FUNCTION_BLOCK CM_Servo EXTENDS CM_Base //IMPLEMENTS I_Servo
VAR_INPUT
	i_refAxis : REFERENCE TO Tc2_MC2.AXIS_REF;
	i_mcHomingMode : Tc2_MC2.MC_HomingMode := Tc2_MC2.MC_HomingMode.MC_Direct;
	i_mcBufferMode : Tc2_MC2.MC_BufferMode := Tc2_MC2.MC_BufferMode.MC_Aborting;
	i_bIclkForward : BOOL := TRUE; //TRUE = interlocked
	i_bIclkBackward : BOOL := TRUE; //TRUE = interlocked
	
	//--i_ref_setting : REFERENCE TO ST_PositioningProfile;
	i_ref_setting : REFERENCE TO ST_SettingsServo;
	
	
	i_ref_eCtrlState : REFERENCE TO E_CtrlState;
END_VAR

VAR
	fbPower : Tc2_MC2.MC_Power;
	fbReset : Tc2_MC2.MC_Reset;
	fbHome : Tc2_MC2.MC_Home;
	fbJog : Tc2_MC2.MC_Jog;
	fbMoveAbsolute : Tc2_MC2.MC_MoveAbsolute;
	fbStop : Tc2_MC2.MC_Stop;

	s_bStaAbsPosBusy : BOOL;
	s_fSetTargetPosition : LREAL;
	
	// Inputs
	I_bEnable AT %I* : BOOL; //Enable from safety controller
	I_bDetReferenceSwitch AT %I* : BOOL; //Reference-/home switch
	I_bDetLimitSwitchPositive AT %I* : BOOL; //Limit switch positive-/CW- direction
	I_bDetLimitSwitchNegative AT %I* : BOOL; //Limit switch negative-/CCW- direction
	
	//Properties
	s_bStatus : BOOL;
	s_bDone : BOOL; 
	s_bBusy : BOOL; 
	s_bActive : BOOL; 
	s_bCommandAborted : BOOL;
	s_bError : BOOL; 
	s_nErrorID : UDINT;
	
	//Requests
	s_bReqNcStop : BOOL;
	s_bReqNcReset : BOOL;
	s_bReqNcHome : BOOL;
	s_bReqNcJog : BOOL;
	s_bReqNcMoveAbs : BOOL;	
	
	// States
	s_bStaEnabled : BOOL;
	s_bStaReferenceSwitch : BOOL;
	s_bStaLimitSwitchPositive : BOOL;
	s_bStaLimitSwitchNegative : BOOL;
	
	s_bStaEnabledControl : BOOL;
	s_bStaEnabledForward : BOOL;
	s_bStaEnabledBackward : BOOL;
	s_bStaReady : BOOL;
	s_bStaHomed : BOOL;
	s_bStaStandstill : BOOL;
	s_bStaMoving : BOOL;
	s_bStaAtPosition : BOOL;
	s_bStaDriveError : BOOL;
	s_bStaWarning : BOOL;
	
	s_bIclkForward : BOOL;
	s_bIclkBackward : BOOL;
	s_sInterlockedReasonForward : STRING; //External interlocked reason for clarifying reason
	s_sInterlockedReasonBackward : STRING; //External interlocked reason for clarifying reason
	
	// Setpoints
	s_fTargetSpeed : LREAL; // Target speed [mm/s]
	
	
	// Alarms
	s_fbAlarmHandlerDriveError : FB_AlarmHandler;
	s_fbAlarmHandlerStartMotorNotAllowed : FB_AlarmHandler;
	s_fbAlarmHandlerMotorForwardInterlocked : FB_AlarmHandler;
	s_fbAlarmHandlerMotorBackwardInterlocked : FB_AlarmHandler;
	
	s_fbAlarmHandlerNotEnabled : FB_AlarmHandler;
	s_fbAlarmHandlerLimitPositiveReached : FB_AlarmHandler;
	s_fbAlarmHandlerLimitNegativeReached : FB_AlarmHandler;
	
	s_errDriveError : BOOL;
	s_wrnMotorForwardInterlocked : BOOL;
	s_wrnMotorBackwardInterlocked : BOOL;
	
	//Hmi
	s_fbHmiBtnHome : FB_HmiBtn;
	s_fbHmiBtnJogPos : FB_HmiBtn;
	s_fbHmiBtnJogNeg : FB_HmiBtn;
	s_fbHmiBtnMoveAbs : FB_HmiBtn;
	//--s_fbHmiBtnPower	: FB_HmiBtn;
	s_fbHmiBtnReset	: FB_HmiBtn;
	s_fbHmiBtnStop: FB_HmiBtn;
	
	s_fbHmiLedEnabledControl : FB_HmiLed;
	s_fbHmiLedEnabledForward : FB_HmiLed;
	s_fbHmiLedEnabledBackward : FB_HmiLed;
	s_fbHmiLedReady : FB_HmiLed;
	s_fbHmiLedHomed : FB_HmiLed;
	s_fbHmiLedStandstill : FB_HmiLed;
	s_fbHmiLedMoving : FB_HmiLed;
	s_fbHmiLedAtPosition : FB_HmiLed;
	s_fbHmiLedDriveError : FB_HmiLed;
	
	//Sequence
	s_eSeqNcTask : E_SeqServo;
	s_fbSeqNcTaskControl : FB_SeqControl;
	s_mcDirection : Tc2_MC2.MC_Direction;
END_VAR


fbPower(
	Axis := i_refAxis,
	Enable := I_bEnable,
	Enable_Positive := I_bDetLimitSwitchPositive,
	Enable_Negative := I_bDetLimitSwitchNegative,
	Override := 100.0,
	BufferMode := TC2_MC2.MC_BufferMode.MC_Aborting,
	Options := ,
	Status => s_bStatus,
	Busy => s_bBusy,
	Active => s_bActive,
	Error => s_bError,
	ErrorID => s_nErrorID);

SUPER^();

METHOD PROTECTED _m_Alarms : BOOL
VAR
	s_bPositiveDirection : BOOL; 
END_VAR

IF NOT SUPER^._m_Alarms() THEN
	RETURN;
END_IF

// Set error bits
s_errDriveError := (i_bReqEnable AND s_bStaDriveError) AND NOT(i_bCmdReset);

// Interlock warnings
s_bPositiveDirection := (i_refAxis.NcToPlc.ActVelo > 0);

IF s_bIclkForward AND NOT(s_bStaStandstill) AND s_bPositiveDirection THEN	
	s_wrnMotorForwardInterlocked := TRUE;
	
	m_Stop(
		i_fDec := i_ref_setting.fStopDec,
		i_fJrk := i_ref_setting.fStopJrk);
	
ELSIF NOT(s_bIclkForward) OR i_bCmdReset THEN
	s_wrnMotorForwardInterlocked := FALSE;
END_IF

IF s_bIclkBackward AND NOT(s_bStaStandstill) AND NOT(s_bPositiveDirection) THEN
	s_wrnMotorBackwardInterlocked := TRUE;
	
	m_Stop(
		i_fDec := i_ref_setting.fStopDec,
		i_fJrk := i_ref_setting.fJogJrk);
		
ELSIF NOT(s_bIclkBackward) OR i_bCmdReset THEN
	s_wrnMotorBackwardInterlocked := FALSE;
END_IF

// Alarm Handlers
s_fbAlarmHandlerDriveError(
	i_bStaActive := s_errDriveError,
	i_sAlarmText := CONCAT(i_sCmName, CONCAT(': Drive - has error: ', UDINT_TO_STRING(i_refAxis.NcToPlc.ErrorCode))));
	
s_fbAlarmHandlerMotorForwardInterlocked(
	i_bStaActive := s_wrnMotorForwardInterlocked,
	i_sAlarmText := CONCAT(i_sCmName, CONCAT(': Motor - interlocked to move forward, Reason: ',CONCAT(s_sInterlockedReasonForward, '.'))));
	
s_fbAlarmHandlerMotorBackwardInterlocked(
	i_bStaActive := s_wrnMotorBackwardInterlocked,
	i_sAlarmText := CONCAT(i_sCmName, CONCAT(': Motor - interlocked to move backward, Reason: ',CONCAT(s_sInterlockedReasonBackward, '.'))));

s_fbAlarmHandlerNotEnabled(
	i_bStaActive := NOT(s_bStaEnabled));
	
s_fbAlarmHandlerLimitPositiveReached(
	i_bStaActive := NOT(s_bStaLimitSwitchPositive));
	
s_fbAlarmHandlerLimitNegativeReached(
	i_bStaActive := NOT(s_bStaLimitSwitchNegative));	
	
// Alarm collector	
s_bStaError := 
	s_fbAlarmHandlerDriveError.q_bStaActive;

// Warning collector
s_bStaWarning := 
	s_fbAlarmHandlerMotorForwardInterlocked.q_bStaActive
	OR s_fbAlarmHandlerMotorBackwardInterlocked.q_bStaActive
	OR s_fbAlarmHandlerNotEnabled.q_bStaActive
	OR s_fbAlarmHandlerLimitPositiveReached.q_bStaActive
	OR s_fbAlarmHandlerLimitNegativeReached.q_bStaActive;
	
_m_Alarms := TRUE;
END_METHOD

METHOD PROTECTED _m_Devices : BOOL
VAR
	sTcDirection : Tc2_MC2.MC_Direction;
END_VAR
IF NOT SUPER^._m_Devices() THEN
	RETURN;
END_IF

s_bStaEnabledControl := s_bStaEnabled AND fbPower.Status;
s_bStaEnabledForward := s_bStaLimitSwitchPositive;
s_bStaEnabledBackward := s_bStaLimitSwitchNegative;

s_bStaReady := i_refAxis.NcToPlc.StateDWord.0;
s_bStaHomed := i_refAxis.NcToPlc.StateDWord.1;
s_bStaStandstill := i_refAxis.NcToPlc.StateDWord.2;
s_bStaMoving := NOT(i_refAxis.NcToPlc.StateDWord.2);
s_bStaAtPosition := i_refAxis.NcToPlc.StateDWord.4;
s_bStaDriveError := i_refAxis.NcToPlc.StateDWord.31;

s_fbSeqNcTaskControl(
	i_nSeqStep := s_eSeqNcTask, 
	i_sStepName := TO_STRING(s_eSeqNcTask), 
	i_bCmdReset := FALSE, 
	i_bStaError := FALSE);

	IF s_bReqNcStop THEN 
		s_eSeqNcTask := E_SeqServo.STOP;
	END_IF		
	
CASE s_eSeqNcTask OF

	E_SeqServo.IDLE:
		
		IF s_bReqNcStop THEN 
			s_eSeqNcTask := E_SeqServo.STOP;
		ELSIF s_bReqNcReset THEN
			s_eSeqNcTask := E_SeqServo.RESET;
		ELSIF s_bReqNcHome THEN
			s_eSeqNcTask := E_SeqServo.HOME;
		ELSIF s_bReqNcJog THEN
			s_eSeqNcTask := E_SeqServo.JOG;
		ELSIF s_bReqNcMoveAbs THEN
			s_eSeqNcTask := E_SeqServo.MOVE_ABS;	
		END_IF
		
	E_SeqServo.STOP:
		IF fbStop.Done THEN
			s_bReqNcStop := FALSE;
			s_eSeqNcTask := E_SeqServo.IDLE;
		END_IF
			
	E_SeqServo.RESET:
		IF fbReset.Done THEN
			s_bReqNcReset := FALSE;
			s_eSeqNcTask := E_SeqServo.IDLE;
		END_IF
			
	E_SeqServo.HOME:
		IF fbHome.Done THEN
			s_bReqNcHome := FALSE;
			s_eSeqNcTask := E_SeqServo.IDLE;
		END_IF
	
	E_SeqServo.JOG:
			IF NOT(s_fbHmiBtnJogPos.p_bStaBtn AND s_fbHmiBtnJogNeg.p_bStaBtn) OR fbJog.Error OR fbJog.CommandAborted THEN
				s_bReqNcJog := FALSE;
				s_eSeqNcTask := E_SeqServo.IDLE;
			END_IF
			
	E_SeqServo.MOVE_ABS:
		IF fbMoveAbsolute.Done OR fbMoveAbsolute.Error OR fbMoveAbsolute.CommandAborted THEN
			s_bReqNcMoveAbs := FALSE;
			s_eSeqNcTask := E_SeqServo.IDLE;
		END_IF
		
END_CASE

fbStop(
	Axis := i_refAxis,
	Execute := s_bReqNcStop,
	Deceleration := i_ref_setting.fStopDec,
	Jerk := i_ref_setting.fStopJrk,
	Options := ,
	Done => s_bDone,
	Busy => s_bBusy,
	Active => s_bActive,
	CommandAborted => s_bCommandAborted,
	Error => s_bError,
	ErrorID => s_nErrorID);

fbReset(
	Axis := i_refAxis,
	Execute := s_bReqNcReset,
	Done => s_bDone,
	Busy => s_bBusy,
	Error => s_bError,
	ErrorID => s_nErrorID);

fbHome(
	Axis := i_refAxis,
	Execute := s_bReqNcHome,
	Position := i_ref_setting.fHomeOffset,
	HomingMode := i_mcHomingMode,
	BufferMode := i_mcBufferMode,
	Options := ,
	bCalibrationCam := I_bDetReferenceSwitch,
	Done => s_bDone,
	Busy => s_bBusy,
	Active => s_bActive,
	CommandAborted => s_bCommandAborted,
	Error => s_bError,
	ErrorID => s_nErrorID);	
	
fbJog(
	Axis := i_refAxis,
	JogForward := s_fbHmiBtnJogPos.p_bStaBtn,
	JogBackwards := s_fbHmiBtnJogNeg.p_bStaBtn,
	Mode := MC_JOGMODE_STANDARD_SLOW,
	Position := ,
	Velocity := i_ref_setting.fJogVel,
	Acceleration := i_ref_setting.fJogAcc,
	Deceleration := i_ref_setting.fJogDec,
	Jerk := i_ref_setting.fJogJrk,
	Done => s_bDone,
	Busy => s_bBusy,
	Active => s_bActive,
	CommandAborted => s_bCommandAborted,
	Error => s_bError,
	ErrorID => s_nErrorID);
	
IF (i_eCtrlMode <> E_CtrlMode.AUTOMATIC) AND (i_eCtrlMode <> E_CtrlMode.MANUAL) THEN
	//--fbMoveAbsolute.Position := i_ref_setting.fAbsPosPos;
	fbMoveAbsolute.Position := s_fSetTargetPosition;
	fbMoveAbsolute.Velocity := i_ref_setting.fAbsPosVel;
	fbMoveAbsolute.Acceleration := i_ref_setting.fAbsPosAcc;
	fbMoveAbsolute.Deceleration := i_ref_setting.fAbsPosDec;
	fbMoveAbsolute.Jerk := i_ref_setting.fAbsPosJrk;
ELSE
	; //positining settings are written from the sequence (this could be different in each case)
END_IF
	
fbMoveAbsolute(
	Axis := i_refAxis,
	Execute := s_bReqNcMoveAbs, 
	Position := ,
	Velocity := ,
	Acceleration := ,
	Deceleration := ,
	Jerk := ,
	BufferMode := i_mcBufferMode,
	Options := ,
	Done => s_bDone,
	Busy => s_bBusy,
	Active => s_bActive,
	CommandAborted => s_bCommandAborted,
	Error => s_bError,
	ErrorID => s_nErrorID);
	
_m_Devices := TRUE;
END_METHOD

METHOD PROTECTED _m_Hmi : BOOL

IF NOT SUPER^._m_Hmi() THEN
	RETURN;
END_IF

//Buttons
s_fbHmiBtnHome();
s_fbHmiBtnJogPos();
s_fbHmiBtnJogNeg();
s_fbHmiBtnMoveAbs();
//--s_fbHmiBtnPower();
s_fbHmiBtnReset();
s_fbHmiBtnStop();

//Leds
s_fbHmiLedEnabledControl(i_bStaLed := s_bStaEnabledControl);
s_fbHmiLedEnabledForward(i_bStaLed := s_bStaEnabledForward);
s_fbHmiLedEnabledBackward(i_bStaLed := s_bStaEnabledBackward);
s_fbHmiLedReady(i_bStaLed := s_bStaReady);
s_fbHmiLedHomed(i_bStaLed := s_bStaHomed);
s_fbHmiLedStandstill(i_bStaLed := s_bStaStandstill);
s_fbHmiLedMoving(i_bStaLed := s_bStaMoving);
s_fbHmiLedAtPosition(i_bStaLed := s_bStaAtPosition);
s_fbHmiLedDriveError(i_bStaLed := s_bStaDriveError);

IF __ISVALIDREF(i_ref_eCtrlState) THEN
	//MAINTENANCE-mode is running
	IF (i_eCtrlMode = E_CtrlMode.MAINTENANCE) AND (i_ref_eCtrlState = E_CtrlState.RUNNING) THEN
		s_fbHmiBtnHome.p_bStaVisible := TRUE;
		s_fbHmiBtnHome.p_bStaEnabled := i_bReqEnable AND s_bStaEnabledControl AND s_bStaStandstill;	

		s_fbHmiBtnJogPos.p_bStaVisible := TRUE;
		s_fbHmiBtnJogPos.p_bStaEnabled := i_bReqEnable AND s_bStaEnabledControl AND s_bStaEnabledForward AND NOT(i_bIclkForward) AND NOT(s_bStaAbsPosBusy);
		
		s_fbHmiBtnJogNeg.p_bStaVisible := TRUE;
		s_fbHmiBtnJogNeg.p_bStaEnabled := i_bReqEnable AND s_bStaEnabledControl AND s_bStaEnabledBackward AND NOT(i_bIclkBackward) AND NOT(s_bStaAbsPosBusy);
	
		s_fbHmiBtnMoveAbs.p_bStaVisible := TRUE;
		s_fbHmiBtnMoveAbs.p_bStaEnabled := i_bReqEnable AND s_bStaEnabledControl AND s_bStaEnabledForward AND s_bStaEnabledBackward AND s_bStaStandstill AND s_bStaHomed AND NOT(i_bIclkForward) AND NOT(i_bIclkBackward);
		
		//--s_fbHmiBtnPower.p_bStaVisible := TRUE;
		//--s_fbHmiBtnPower.p_bStaEnabled := TRUE;
		
		s_fbHmiBtnReset.p_bStaVisible := TRUE;
		s_fbHmiBtnReset.p_bStaEnabled := TRUE;
		
		s_fbHmiBtnStop.p_bStaVisible := TRUE;
		s_fbHmiBtnStop.p_bStaEnabled := TRUE;
		
		//Maintenance commands from buttons
		IF s_fbHmiBtnStop.p_osrBtnPress THEN
			s_bReqNcStop := TRUE;
		END_IF
		
		IF s_fbHmiBtnReset.p_osrBtnPress THEN
			s_bReqNcReset := TRUE;
		END_IF
		
		IF s_fbHmiBtnHome.p_osrBtnPress THEN
			s_bReqNcHome := TRUE;
		END_IF
		
		IF s_fbHmiBtnJogNeg.p_osrBtnPress THEN
			s_mcDirection := Tc2_MC2.MC_Direction.MC_Negative_Direction;
			s_bReqNcJog := TRUE;
		END_IF
		
		IF s_fbHmiBtnJogPos.p_osrBtnPress THEN
			s_mcDirection := Tc2_MC2.MC_Direction.MC_Positive_Direction;
			s_bReqNcJog := TRUE;
		END_IF
		
		IF s_fbHmiBtnMoveAbs.p_osrBtnPress THEN
			s_bReqNcMoveAbs := TRUE;
		END_IF
		
	//other-mode	
	ELSE
		s_fbHmiBtnHome.p_bStaVisible := FALSE;
		s_fbHmiBtnHome.p_bStaEnabled := FALSE;
		
		s_fbHmiBtnJogPos.p_bStaVisible := FALSE;
		s_fbHmiBtnJogPos.p_bStaEnabled := FALSE;
		
		s_fbHmiBtnJogNeg.p_bStaVisible := FALSE;
		s_fbHmiBtnJogNeg.p_bStaEnabled := FALSE;
		
		s_fbHmiBtnMoveAbs.p_bStaVisible := FALSE;
		s_fbHmiBtnMoveAbs.p_bStaEnabled := FALSE;
		
		//--s_fbHmiBtnPower.p_bStaVisible := FALSE;
		//--s_fbHmiBtnPower.p_bStaEnabled := FALSE;
		
		s_fbHmiBtnReset.p_bStaVisible := FALSE;
		s_fbHmiBtnReset.p_bStaEnabled := FALSE;
		
		s_fbHmiBtnStop.p_bStaVisible := FALSE;
		s_fbHmiBtnStop.p_bStaEnabled := FALSE;
	END_IF
END_IF
	
_m_Hmi := TRUE;
END_METHOD

METHOD PROTECTED _m_Init : BOOL

IF NOT SUPER^._m_Init() THEN
	RETURN;
END_IF

//Alarm Config
// Alarm Handlers
s_fbAlarmHandlerDriveError.i_eAlarmLevel := E_AlarmLevel.Alarm;
s_fbAlarmHandlerMotorForwardInterlocked.i_eAlarmLevel := E_AlarmLevel.Warning;
s_fbAlarmHandlerMotorBackwardInterlocked.i_eAlarmLevel := E_AlarmLevel.Warning;
s_fbAlarmHandlerNotEnabled.i_eAlarmLevel := E_AlarmLevel.Warning;
s_fbAlarmHandlerNotEnabled.i_sAlarmText := CONCAT(i_sCmName, ' - Not enabled');
s_fbAlarmHandlerLimitPositiveReached.i_eAlarmLevel := E_AlarmLevel.Warning;
s_fbAlarmHandlerLimitPositiveReached.i_sAlarmText := CONCAT(i_sCmName, ' - Limits witch positvie reached');
s_fbAlarmHandlerLimitNegativeReached.i_eAlarmLevel := E_AlarmLevel.Warning;
s_fbAlarmHandlerLimitNegativeReached.i_sAlarmText := CONCAT(i_sCmName, ' - Limits witch negative reached');

//Hmi 
	//Buttons
	s_fbHmiBtnHome.p_eButtontype := E_HmiButtonType.PUSHBUTTON;
	s_fbHmiBtnHome.p_bStaVisible := FALSE;
	s_fbHmiBtnHome.p_bStaEnabled := FALSE;		
	s_fbHmiBtnHome.p_sBtnText := 'Home';
	
	s_fbHmiBtnJogPos.p_eButtontype := E_HmiButtonType.PUSHBUTTON;
	s_fbHmiBtnJogPos.p_bStaVisible := FALSE;
	s_fbHmiBtnJogPos.p_bStaEnabled := FALSE;		
	s_fbHmiBtnJogPos.p_sBtnText := 'Jog Positive';
	
	s_fbHmiBtnJogNeg.p_eButtontype := E_HmiButtonType.PUSHBUTTON;
	s_fbHmiBtnJogNeg.p_bStaVisible := FALSE;
	s_fbHmiBtnJogNeg.p_bStaEnabled := FALSE;		
	s_fbHmiBtnJogNeg.p_sBtnText := 'Jog Negative';
	
	s_fbHmiBtnMoveAbs.p_eButtontype := E_HmiButtonType.PUSHBUTTON;
	s_fbHmiBtnMoveAbs.p_bStaVisible := FALSE;
	s_fbHmiBtnMoveAbs.p_bStaEnabled := FALSE;		
	s_fbHmiBtnMoveAbs.p_sBtnText := 'Move Absolute';
	
	//--s_fbHmiBtnPower.p_eButtontype := E_HmiButtonType.PUSHBUTTON;
	//--s_fbHmiBtnPower.p_bStaVisible := FALSE;
	//--s_fbHmiBtnPower.p_bStaEnabled := FALSE;		
	//--s_fbHmiBtnPower.p_sBtnText := 'Enable';

	s_fbHmiBtnReset.p_eButtontype := E_HmiButtonType.PUSHBUTTON;
	s_fbHmiBtnReset.p_bStaVisible := FALSE;
	s_fbHmiBtnReset.p_bStaEnabled := FALSE;		
	s_fbHmiBtnReset.p_sBtnText := 'Reset';
	
	s_fbHmiBtnReset.p_eButtontype := E_HmiButtonType.PUSHBUTTON;
	s_fbHmiBtnReset.p_bStaVisible := FALSE;
	s_fbHmiBtnReset.p_bStaEnabled := FALSE;		
	s_fbHmiBtnReset.p_sBtnText := 'Reset';
	
	s_fbHmiBtnStop.p_eButtontype := E_HmiButtonType.PUSHBUTTON;
	s_fbHmiBtnStop.p_bStaVisible := FALSE;
	s_fbHmiBtnStop.p_bStaEnabled := FALSE;		
	s_fbHmiBtnStop.p_sBtnText := 'Stop';
	
	//Leds
	s_fbHmiLedEnabledControl.p_bStaVisible := FALSE;
	s_fbHmiLedEnabledControl.p_sToHmiDescriptionLed := 'Enabled Control';
	
	s_fbHmiLedEnabledForward.p_bStaVisible := FALSE;
	s_fbHmiLedEnabledForward.p_sToHmiDescriptionLed := 'Enabled Forward';
	
	s_fbHmiLedEnabledBackward.p_bStaVisible := FALSE;
	s_fbHmiLedEnabledBackward.p_sToHmiDescriptionLed := 'Enabled Backward';
	
	s_fbHmiLedReady.p_bStaVisible := FALSE;
	s_fbHmiLedReady.p_sToHmiDescriptionLed := 'Ready';
	
	s_fbHmiLedHomed.p_bStaVisible := FALSE;
	s_fbHmiLedHomed.p_sToHmiDescriptionLed := 'Homed';
	
	s_fbHmiLedStandstill.p_bStaVisible := FALSE;
	s_fbHmiLedStandstill.p_sToHmiDescriptionLed := 'Standstill';
	
	s_fbHmiLedMoving.p_bStaVisible := FALSE;
	s_fbHmiLedMoving.p_sToHmiDescriptionLed := 'Moving';

	s_fbHmiLedAtPosition.p_bStaVisible := FALSE;
	s_fbHmiLedAtPosition.p_sToHmiDescriptionLed := 'At Position';
	
	s_fbHmiLedDriveError.p_bStaVisible := FALSE;
	s_fbHmiLedDriveError.p_sToHmiDescriptionLed := 'Drive Error';
	
_m_Init := TRUE;
END_METHOD

METHOD PROTECTED _m_Inputs : BOOL

IF NOT SUPER^._m_Inputs() THEN
	RETURN;
END_IF

s_bReqNcReset := i_bCmdReset; 

s_bStaEnabled := I_bEnable;
s_bStaReferenceSwitch := I_bDetReferenceSwitch;
s_bStaLimitSwitchPositive := I_bDetLimitSwitchPositive;
s_bStaLimitSwitchNegative := I_bDetLimitSwitchNegative;

s_bIclkForward := i_bIclkForward;
s_bIclkBackward := i_bIclkBackward;

//Local reasons, first
IF NOT(s_bStaEnabled) AND (i_eCtrlMode = E_CtrlMode.MAINTENANCE) THEN  
	s_sInterlockedReasonForward := 'Not enabled';
ELSIF NOT(s_bStaLimitSwitchPositive) THEN  
	s_sInterlockedReasonForward := 'Limit-switch forward';
ELSE
	;// Else, allow external to write
END_IF

//Local reasons, first
IF NOT(s_bStaEnabled) AND (i_eCtrlMode = E_CtrlMode.MAINTENANCE) THEN  
	s_sInterlockedReasonBackward := 'Not enabled';
ELSIF NOT(s_bStaLimitSwitchNegative) THEN  
	s_sInterlockedReasonBackward := 'Limit-switch backward';
ELSE
	;// Else, allow external to write
END_IF

_m_Inputs := TRUE;
END_METHOD

METHOD PROTECTED _m_Outputs : BOOL

IF NOT SUPER^._m_Outputs() THEN
	RETURN;
END_IF

_m_Outputs := TRUE;
END_METHOD

//Returms TRUE if move absolute is done
METHOD PUBLIC m_MoveAbsolute : BOOL
VAR_INPUT
	i_stPositioningProfile : ST_PositioningProfile;
END_VAR
VAR_OUTPUT
	o_Busy : BOOL;
	o_bDone : BOOL;
	o_bError : BOOL;
END_VAR

s_bReqNcMoveAbs := TRUE;

//Inputs
fbMoveAbsolute.Position := i_stPositioningProfile.fPos;
fbMoveAbsolute.Velocity := i_stPositioningProfile.fVel;
fbMoveAbsolute.Acceleration := i_stPositioningProfile.fAcc;
fbMoveAbsolute.Deceleration := i_stPositioningProfile.fDec;
fbMoveAbsolute.Jerk := i_stPositioningProfile.fJrk;

//Outputs
o_Busy := fbMoveAbsolute.Busy;
o_bDone := fbMoveAbsolute.Done;
o_bError := fbMoveAbsolute.Error;
	
m_MoveAbsolute := s_bDone;
END_METHOD

//Returms TRUE if reset is done
METHOD PUBLIC m_Reset : BOOL
VAR_OUTPUT
	o_Busy : BOOL;
	o_bDone : BOOL;
	o_bError : BOOL;
END_VAR

s_bReqNcReset := TRUE;

//Outputs
o_Busy := fbReset.Busy;
o_bDone := fbReset.Done;
o_bError := fbReset.Error;
	
m_Reset := s_bDone;
END_METHOD

//Returms TRUE if stop is done
METHOD PUBLIC m_Stop : BOOL
VAR_INPUT
	i_fDec : LREAL; 
	i_fJrk : LREAL;
END_VAR
VAR_OUTPUT
	o_Busy : BOOL;
	o_bDone : BOOL;
	o_bError : BOOL;
END_VAR

s_bReqNcStop := TRUE;

//Inputs
fbStop.Deceleration := i_fDec;
fbStop.Jerk := i_fJrk;

//Outputs
o_Busy := fbStop.Busy;
o_bDone := fbStop.Done;
o_bError := fbStop.Error;
	
m_Stop := s_bDone;
END_METHOD

PROPERTY PUBLIC p_bActive : BOOL
GET

p_bActive := s_bActive;
END_GET
END_PROPERTY

PROPERTY PUBLIC p_bAtPosition : BOOL
GET

p_bAtPosition := s_bStaAtPosition;
END_GET
END_PROPERTY

PROPERTY PUBLIC p_bBusy : BOOL
GET

p_bBusy := s_bBusy;
END_GET
END_PROPERTY

PROPERTY PUBLIC p_bCommandAborted : BOOL
GET

p_bCommandAborted := s_bCommandAborted;
END_GET
END_PROPERTY

PROPERTY PUBLIC p_bDone : BOOL
GET

p_bDone := s_bDone;
END_GET
END_PROPERTY

PROPERTY PUBLIC p_bError : BOOL
GET

p_bError := s_bStaError;
END_GET
END_PROPERTY

PROPERTY PUBLIC p_bHomed : BOOL
GET

p_bHomed := i_refAxis.Status.Homed;
END_GET
END_PROPERTY

PROPERTY PUBLIC p_bStandstill : BOOL
GET

p_bStandstill := i_refAxis.Status.StandStill;
END_GET
END_PROPERTY

PROPERTY PUBLIC p_bWarning : BOOL
GET

p_bWarning := s_bStaWarning;
END_GET
END_PROPERTY

PROPERTY PUBLIC p_fPosition : LREAL
GET

p_fPosition := i_refAxis.NcToPlc.ActPos;
END_GET
END_PROPERTY

PROPERTY PUBLIC p_fSetTargetPosition : LREAL
GET

p_fSetTargetPosition := s_fSetTargetPosition;
END_GET
SET

s_fSetTargetPosition := p_fSetTargetPosition;
END_SET
END_PROPERTY

PROPERTY PUBLIC p_fVelocity : LREAL
GET

p_fVelocity := i_refAxis.NcToPlc.ActVelo;
END_GET
END_PROPERTY

PROPERTY PUBLIC p_nErrorID : UDINT
GET

p_nErrorID := s_nErrorID;
END_GET
END_PROPERTY

{attribute 'monitoring':='call'}
PROPERTY PUBLIC p_sInterlockedReasonBackward : STRING(GVL.g_MAX_LEN_INTERLOCK_REASON)
GET

p_sInterlockedReasonBackward := s_sInterlockedReasonBackward;
END_GET
SET

s_sInterlockedReasonBackward := p_sInterlockedReasonBackward;
END_SET
END_PROPERTY

{attribute 'monitoring':='call'}
PROPERTY PUBLIC p_sInterlockedReasonForward : STRING(GVL.g_MAX_LEN_INTERLOCK_REASON)
GET

p_sInterlockedReasonForward := s_sInterlockedReasonForward;
END_GET
SET

s_sInterlockedReasonForward := p_sInterlockedReasonForward;
END_SET
END_PROPERTY

END_FUNCTION_BLOCK

(* stored: Version 1.1.0.1, ProductVersion 3.1.4024.12
   POU CM_Servo: Id {29dfdbae-f16d-497a-b262-2baea4701d77}, SpecialFunc None
   Folder Methods: Id {c7dc02dc-f2cb-44e5-89eb-2e4085b6a909}
   Folder Base: Id {1f8bf144-7c2c-4c0f-9741-6defd5a25c8d}
   Folder Properties: Id {c3e008a7-9dfe-49e0-9cc5-18c79327535a}
   Method _m_Alarms: Id {c522f959-6f84-4a96-b11e-07b34d6dcd1a}
   Method _m_Devices: Id {9e243b00-6ff1-489e-8f7b-4b8502bb7008}
   Method _m_Hmi: Id {d347e6d1-38a6-4faa-8926-d4b86b27fe7e}
   Method _m_Init: Id {04dfb054-6b11-4b5e-a48d-10fd0c5ab89c}
   Method _m_Inputs: Id {6f1bac9d-85af-4aa0-99cc-0441d85b988e}
   Method _m_Outputs: Id {705beffa-2023-4b46-ae05-94ae1d9439ab}
   Method m_MoveAbsolute: Id {33b1db53-3e9c-45b9-acb8-f86fe15b34c1}
   Method m_Reset: Id {3c0e8a28-dc02-4569-b874-5e16ba6f1cc1}
   Method m_Stop: Id {8221ae9d-4a4c-432f-85a4-2df50a225ff5}
   Property p_bActive: Id {fdebd466-4355-4961-86f7-17cb1e74e332}
   Get Get: Id {12554b68-dea8-473b-b98f-bf82edb9ad16}
   Property p_bAtPosition: Id {1427e9eb-62b0-446d-9229-ecc0728aa739}
   Get Get: Id {f7ed9d8f-2a48-406a-a4f6-3a1e43916f46}
   Property p_bBusy: Id {a6bb4214-9e42-46dd-a8f3-995e364772d0}
   Get Get: Id {7080bc48-c94e-419b-9e7d-df95694c753e}
   Property p_bCommandAborted: Id {32bd9d7d-f5a3-4f89-9a59-0294a826c560}
   Get Get: Id {a39acfdd-fde9-4118-9e65-bd86ad5a94af}
   Property p_bDone: Id {09a3960b-0e70-4e33-a3d6-ff5a57122d42}
   Get Get: Id {e656286c-fa2b-43ef-a794-1f2819d97be9}
   Property p_bError: Id {7759aec3-bd8b-4f0c-9913-656b2c70cf6a}
   Get Get: Id {67b5f8fe-c6e4-4145-9f0e-f9d36c480d63}
   Property p_bHomed: Id {29d86fc1-be45-4333-91ce-9bdc79739fba}
   Get Get: Id {3bff5f71-c84f-4863-9be2-8ae02d95a4db}
   Property p_bStandstill: Id {06fe4adf-3a6b-49c2-a8e8-c5de29d0c1af}
   Get Get: Id {e4db3dbb-9fbf-4ca7-ba91-332924a328ae}
   Property p_bWarning: Id {b8faca11-510c-4a1a-b235-b64a1404f723}
   Get Get: Id {209789e2-4f7f-40c8-b8a3-6199664c8d00}
   Property p_fPosition: Id {e5ef2cba-1955-4270-98db-4d1260096b27}
   Get Get: Id {440682b1-07c0-42c1-8793-ae28db2834f6}
   Property p_fSetTargetPosition: Id {d8bd5c56-1afd-4449-9ff5-408d5b4dc1a6}
   Get Get: Id {2f75fc55-e4e2-4d1a-9e2e-5f2488ab159d}
   Set Set: Id {8e420d50-b498-4fbd-a8d3-bcf62048045f}
   Property p_fVelocity: Id {e4d08808-aacd-469e-bccf-b788a2ac516e}
   Get Get: Id {a4e61425-56d9-43cd-b7a5-921c2a97d144}
   Property p_nErrorID: Id {063f18f8-6320-4761-b8fc-9920f5ec0c3a}
   Get Get: Id {fa545b5b-0766-4028-bde3-78e42d22c7e0}
   Property p_sInterlockedReasonBackward: Id {2cbc61be-2980-49ea-9737-516b9cc082cc}
   Get Get: Id {6302c11b-5d35-483e-93f6-02d7e278d314}
   Set Set: Id {736eeda3-1c6b-466b-a8c9-83add0319e61}
   Property p_sInterlockedReasonForward: Id {54c2d2dd-7915-4fa3-818c-250a80b85813}
   Get Get: Id {c021f6d7-6c1d-45d2-8cf8-029294050c22}
   Set Set: Id {ae73b161-60cd-49c4-958c-4f84879e0c7c} *)
